FUNCTION_BLOCK FB_HNLTSystem
VAR_INPUT
END_VAR
VAR_OUTPUT
END_VAR
VAR
	
	// heat counters
	WMZ246 : FB_MollineC3HeatCounter;
	WMZ247 : FB_MollineC3HeatCounter;

END_VAR

WMZ246(aHeatCounterTelegramm := MBus.Telegramm_WMZ_246);
WMZ247(aHeatCounterTelegramm := MBus.Telegramm_WMZ_247);

END_FUNCTION_BLOCK

(* stored: Version 1.1.0.1, ProductVersion 3.1.4024.6
   POU FB_HNLTSystem: Id {ad378e4f-4dcc-4fbd-a624-889931407b46}, SpecialFunc None *)
